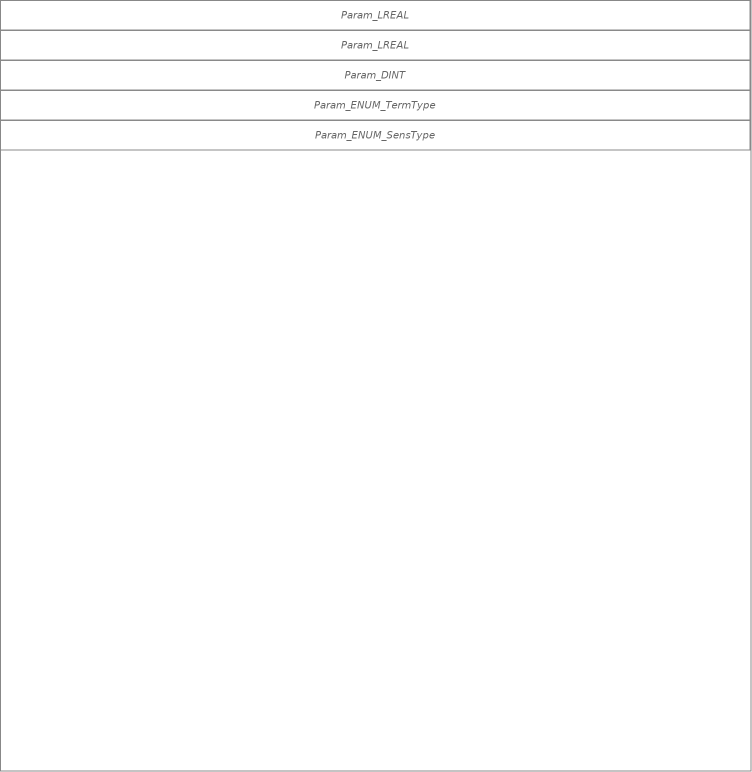
VISUALIZATION Visu_Mparam_Temperatur  // 752x772
    Frame (0,0 750x30)
        shows Param_LREAL(nIdx := GlobalOne)
    Frame (0,30 750x30)
        shows Param_LREAL(nIdx := 2)
    Frame (0,60 750x30)
        shows Param_DINT(nIdx := 9)
    Frame (0,90 750x30)
        shows Param_ENUM_TermType(nIdx := 3)
    Frame (0,120 750x30)
        shows Param_ENUM_SensType(nIdx := 4)
    Rectangle (0,740 750x30)
END_VISUALIZATION

(* stored: Version 1.1.0.1, ProductVersion 3.1.4024.12
   Visu Visu_Mparam_Temperatur: Id {7e063f9a-a9b4-4a7c-a542-247d043c874b} *)
